// TIA Portal V17 export
// export: Created 2024-09-26T08:53:41.1768977Z, ExportSetting WithDefaults, DisplayName Totally Integrated Automation Portal, DisplayVersion V17, DisplayName TIA Portal Openness, DisplayVersion V17, DisplayName TIA Portal Version Control Interface, DisplayVersion V17, DisplayName STEP 7 Professional, DisplayVersion V17, DisplayName STEP 7 Safety, DisplayVersion V17, DisplayName WinCC Advanced / Unified PC, DisplayVersion V17
DATA_BLOCK "SMA_Flow_1_DB"   // DB5
VERSION : 0.1
// stored: AutoNumber true, DBAccessibleFromOPCUA true, InstanceOfName SMA_Flow_1, InstanceOfType FB
"SMA_Flow_1"
   // VAR_INPUT
   //    bRun : Bool;
   //    tDutyCycle : Time;
   //    rFlow_Input : Real;
   // END_VAR
   // VAR_OUTPUT
   //    Flow { ExternalAccessible := 'False'; ExternalVisible := 'False'; ExternalWritable := 'False'} : Real;
   // END_VAR
BEGIN
END_DATA_BLOCK
